Yaskawa INFORM job: MALBEN3.JBI

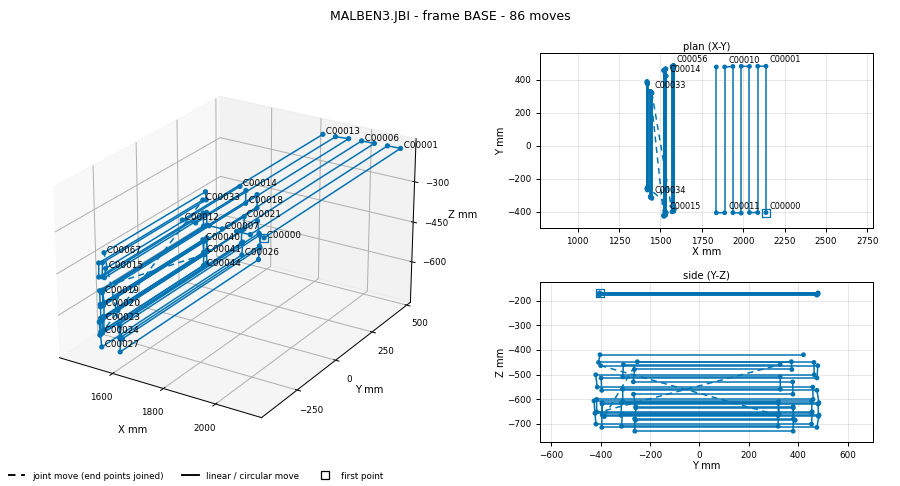
[picture p0: tool path of MALBEN3.JBI in frame BASE, 86 of 92 moves have a stored position in this frame; points joined in program order, loops and branches not executed]
/JOB
//NAME MALBEN3
//POS
///NPOS 86,0,86,0,0,0
///TOOL 0
///POSTYPE BASE
///RECTAN
///RCONF 1,0,0,0,0,0,0,0,0,0,0,0,0,0,0,0,0,0,0,0,0,0,0,0
C00000=2138.089252,-404.380452,-169.043680,175.000000,5.000000,5.000000
C00001=2138.089252,480.563343,-169.043680,175.000000,5.000000,5.000000
C00002=2088.089252,480.435732,-170.096495,175.000000,5.000000,5.000000
C00003=2088.089252,-404.293829,-170.096495,175.000000,5.000000,5.000000
C00004=2038.089252,-404.161569,-171.304879,175.000000,5.000000,5.000000
C00005=2038.089252,479.548369,-171.304879,175.000000,5.000000,5.000000
C00006=1988.089252,480.242625,-172.720240,175.000000,5.000000,5.000000
C00007=1988.089252,-407.599887,-172.720240,175.000000,5.000000,5.000000
C00008=1938.089252,-404.906531,-174.491375,175.000000,5.000000,5.000000
C00009=1938.089252,479.135112,-174.491375,175.000000,5.000000,5.000000
C00010=1888.089252,475.934269,-176.316370,175.000000,5.000000,5.000000
C00011=1888.089252,-405.530643,-176.316370,175.000000,5.000000,5.000000
C00012=1837.950754,-405.573743,-177.808492,175.000000,5.000000,5.000000
C00013=1837.950754,475.917367,-177.808492,175.000000,5.000000,5.000000
C00014=1534.901840,421.478015,-419.338167,175.000000,-89.999999,5.000000
C00015=1534.901840,-402.937946,-419.338167,175.000000,-89.999999,5.000000
C00016=1533.144001,-408.647490,-450.491085,175.000000,-89.999999,5.000000
C00017=1533.144001,464.153807,-450.491085,175.000000,-89.999999,5.000000
C00018=1531.375428,464.936799,-500.491085,175.000000,-89.999999,5.000000
C00019=1531.375428,-420.046716,-500.491085,175.000000,-89.999999,5.000000
C00020=1529.352914,-413.942085,-550.491085,175.000000,-89.999999,5.000000
C00021=1529.352914,459.233172,-550.491085,175.000000,-89.999999,5.000000
C00022=1526.912057,460.521115,-600.491085,175.000000,-89.999999,5.000000
C00023=1526.912057,-416.386557,-600.491085,175.000000,-89.999999,5.000000
C00024=1524.500347,-416.295497,-650.491085,175.000000,-89.999999,5.000000
C00025=1524.500347,456.784052,-650.491085,175.000000,-89.999999,5.000000
C00026=1522.504336,454.310846,-700.491085,175.000000,-89.999999,5.000000
C00027=1522.504336,-419.163579,-700.491085,175.000000,-89.999999,5.000000
C00028=1520.880267,-427.203082,-606.153518,180.000000,-60.000000,0.000000
C00029=1520.880267,455.493151,-606.153518,180.000000,-60.000000,0.000000
C00030=1519.374249,455.436528,-656.153518,180.000000,-60.000000,0.000000
C00031=1519.374249,-422.503865,-656.153518,180.000000,-60.000000,0.000000
C00032=1519.374249,-422.503865,-656.153518,180.000000,-60.000000,0.000000
C00033=1438.715086,327.474473,-459.345178,175.000000,-89.999999,5.000000
C00034=1438.715086,-307.755951,-459.345178,175.000000,-89.999999,5.000000
C00035=1439.798940,-310.872345,-509.345178,175.000000,-89.999999,5.000000
C00036=1439.798940,327.369569,-509.345178,175.000000,-89.999999,5.000000
C00037=1441.037287,327.734598,-559.345178,175.000000,-89.999999,5.000000
C00038=1441.037287,-310.730484,-559.345178,175.000000,-89.999999,5.000000
C00039=1442.396814,-310.620464,-609.345178,175.000000,-89.999999,5.000000
C00040=1442.396814,320.382842,-609.345178,175.000000,-89.999999,5.000000
C00041=1443.632843,322.978132,-659.345178,175.000000,-89.999999,5.000000
C00042=1443.632843,-311.906310,-659.345178,175.000000,-89.999999,5.000000
C00043=1445.183093,-315.667760,-709.345178,175.000000,-89.999999,5.000000
C00044=1445.183093,319.105240,-709.345178,175.000000,-89.999999,5.000000
C00045=1446.831419,319.750011,-615.007611,180.000000,-60.000000,0.000000
C00046=1446.831419,-315.758164,-615.007611,180.000000,-60.000000,0.000000
C00047=1448.220568,-317.504562,-665.007611,180.000000,-60.000000,0.000000
C00048=1448.220568,318.562813,-665.007611,180.000000,-60.000000,0.000000
C00049=1448.220568,318.562813,-665.007611,180.000000,-60.000000,0.000000
C00050=1570.356830,-399.922593,-463.648284,175.000000,-89.999999,5.000000
C00051=1570.356830,479.704633,-463.648284,175.000000,-89.999999,5.000000
C00052=1572.586404,476.504213,-513.648284,175.000000,-89.999999,5.000000
C00053=1572.586404,-398.280973,-513.648284,175.000000,-89.999999,5.000000
C00054=1574.691641,-395.744807,-563.648284,175.000000,-89.999999,5.000000
C00055=1574.691641,476.324205,-563.648284,175.000000,-89.999999,5.000000
C00056=1576.436703,484.068766,-613.648284,175.000000,-89.999999,5.000000
C00057=1576.436703,-394.544332,-613.648284,175.000000,-89.999999,5.000000
C00058=1578.039943,-393.977688,-663.648284,175.000000,-89.999999,5.000000
C00059=1578.039943,484.690765,-663.648284,175.000000,-89.999999,5.000000
C00060=1579.649911,475.998417,-713.648284,175.000000,-89.999999,5.000000
C00061=1579.649911,-395.540713,-713.648284,175.000000,-89.999999,5.000000
C00062=1580.841793,-394.570108,-619.310716,180.000000,-60.000000,0.000000
C00063=1580.841793,480.898770,-619.310716,180.000000,-60.000000,0.000000
C00064=1582.269908,482.315169,-669.310716,180.000000,-60.000000,0.000000
C00065=1582.269908,-385.635636,-669.310716,180.000000,-60.000000,0.000000
C00066=1582.269908,-385.635636,-669.310716,180.000000,-60.000000,0.000000
C00067=1420.964910,-251.559719,-447.665037,175.000000,-89.999999,5.000000
C00068=1420.964910,372.604123,-447.665037,175.000000,-89.999999,5.000000
C00069=1422.373131,374.697923,-479.185471,175.000000,-89.999999,5.000000
C00070=1422.373131,-263.019191,-479.185471,175.000000,-89.999999,5.000000
C00071=1421.975445,-267.696341,-529.185471,175.000000,-89.999999,5.000000
C00072=1421.975445,377.834218,-529.185471,175.000000,-89.999999,5.000000
C00073=1421.594266,378.934991,-579.185471,175.000000,-89.999999,5.000000
C00074=1421.594266,-266.992153,-579.185471,175.000000,-89.999999,5.000000
C00075=1420.418300,-258.080778,-629.185471,175.000000,-89.999999,5.000000
C00076=1420.418300,379.690351,-629.185471,175.000000,-89.999999,5.000000
C00077=1419.981840,380.884372,-679.185471,175.000000,-89.999999,5.000000
C00078=1419.981840,-262.435258,-679.185471,175.000000,-89.999999,5.000000
C00079=1419.737986,-261.680466,-729.185471,175.000000,-89.999999,5.000000
C00080=1419.737986,379.769100,-729.185471,175.000000,-89.999999,5.000000
C00081=1419.270374,380.316359,-634.847904,180.000000,-60.000000,0.000000
C00082=1419.270374,-257.794213,-634.847904,180.000000,-60.000000,0.000000
C00083=1418.737426,-258.418231,-684.847904,180.000000,-60.000000,0.000000
C00084=1418.737426,387.426469,-684.847904,180.000000,-60.000000,0.000000
C00085=1418.737426,387.426469,-684.847904,180.000000,-60.000000,0.000000
///POSTYPE PULSE
///PULSE
EC00000=0
EC00001=0
EC00002=0
EC00003=0
EC00004=0
EC00005=0
EC00006=0
EC00007=0
EC00008=0
EC00009=0
EC00010=0
EC00011=0
EC00012=0
EC00013=0
EC00014=0
EC00015=0
EC00016=0
EC00017=0
EC00018=0
EC00019=0
EC00020=0
EC00021=0
EC00022=0
EC00023=0
EC00024=0
EC00025=0
EC00026=0
EC00027=0
EC00028=0
EC00029=0
EC00030=0
EC00031=0
EC00032=92160
EC00033=92160
EC00034=92160
EC00035=92160
EC00036=92160
EC00037=92160
EC00038=92160
EC00039=92160
EC00040=92160
EC00041=92160
EC00042=92160
EC00043=92160
EC00044=92160
EC00045=92160
EC00046=92160
EC00047=92160
EC00048=92160
EC00049=184320
EC00050=184320
EC00051=184320
EC00052=184320
EC00053=184320
EC00054=184320
EC00055=184320
EC00056=184320
EC00057=184320
EC00058=184320
EC00059=184320
EC00060=184320
EC00061=184320
EC00062=184320
EC00063=184320
EC00064=184320
EC00065=184320
EC00066=276480
EC00067=276480
EC00068=276480
EC00069=276480
EC00070=276480
EC00071=276480
EC00072=276480
EC00073=276480
EC00074=276480
EC00075=276480
EC00076=276480
EC00077=276480
EC00078=276480
EC00079=276480
EC00080=276480
EC00081=276480
EC00082=276480
EC00083=276480
EC00084=276480
EC00085=368640
//INST
///DATE 2023/03/16 10:48
///ATTR SC,RW,RJ
////FRAME BASE
///GROUP1 RB1,ST1
NOP
MOVJ P009 EX000 VJ=15.00
MOVJ C00000 EC00000 VJ=15.0
CALL JOB:SPYON
MOVL C00001 EC00001 V=300.0
MOVL C00002 EC00002 V=300.0
MOVL C00003 EC00003 V=300.0
MOVL C00004 EC00004 V=300.0
MOVL C00005 EC00005 V=300.0
MOVL C00006 EC00006 V=300.0
MOVL C00007 EC00007 V=300.0
MOVL C00008 EC00008 V=300.0
MOVL C00009 EC00009 V=300.0
MOVL C00010 EC00010 V=300.0
MOVL C00011 EC00011 V=300.0
MOVL C00012 EC00012 V=300.0
MOVL C00013 EC00013 V=300.0
CALL JOB:SPYOF
MOVJ P009 VJ=15.00
MOVJ C00014 EC00014 VJ=15.0
CALL JOB:SPYON
MOVL C00015 EC00015 V=300.0
MOVL C00016 EC00016 V=300.0
MOVL C00017 EC00017 V=300.0
MOVL C00018 EC00018 V=300.0
MOVL C00019 EC00019 V=300.0
MOVL C00020 EC00020 V=300.0
MOVL C00021 EC00021 V=300.0
MOVL C00022 EC00022 V=300.0
MOVL C00023 EC00023 V=300.0
MOVL C00024 EC00024 V=300.0
MOVL C00025 EC00025 V=300.0
MOVL C00026 EC00026 V=300.0
MOVL C00027 EC00027 V=300.0
MOVL C00028 EC00028 V=300.0
MOVL C00029 EC00029 V=300.0
MOVL C00030 EC00030 V=300.0
MOVL C00031 EC00031 V=300.0
CALL JOB:SPYOF
MOVJ P009 VJ=15.00
MOVL C00032 EC00032 V=300.0
MOVJ C00033 EC00033 VJ=15.0
CALL JOB:SPYON
MOVL C00034 EC00034 V=300.0
MOVL C00035 EC00035 V=300.0
MOVL C00036 EC00036 V=300.0
MOVL C00037 EC00037 V=300.0
MOVL C00038 EC00038 V=300.0
MOVL C00039 EC00039 V=300.0
MOVL C00040 EC00040 V=300.0
MOVL C00041 EC00041 V=300.0
MOVL C00042 EC00042 V=300.0
MOVL C00043 EC00043 V=300.0
MOVL C00044 EC00044 V=300.0
MOVL C00045 EC00045 V=300.0
MOVL C00046 EC00046 V=300.0
MOVL C00047 EC00047 V=300.0
MOVL C00048 EC00048 V=300.0
CALL JOB:SPYOF
MOVJ P009 VJ=15.00
MOVL C00049 EC00049 V=300.0
MOVJ C00050 EC00050 VJ=15.0
CALL JOB:SPYON
MOVL C00051 EC00051 V=300.0
MOVL C00052 EC00052 V=300.0
MOVL C00053 EC00053 V=300.0
MOVL C00054 EC00054 V=300.0
MOVL C00055 EC00055 V=300.0
MOVL C00056 EC00056 V=300.0
MOVL C00057 EC00057 V=300.0
MOVL C00058 EC00058 V=300.0
MOVL C00059 EC00059 V=300.0
MOVL C00060 EC00060 V=300.0
MOVL C00061 EC00061 V=300.0
MOVL C00062 EC00062 V=300.0
MOVL C00063 EC00063 V=300.0
MOVL C00064 EC00064 V=300.0
MOVL C00065 EC00065 V=300.0
CALL JOB:SPYOF
MOVJ P009 VJ=15.00
MOVL C00066 EC00066 V=300.0
MOVJ C00067 EC00067 VJ=15.0
CALL JOB:SPYON
MOVL C00068 EC00068 V=300.0
MOVL C00069 EC00069 V=300.0
MOVL C00070 EC00070 V=300.0
MOVL C00071 EC00071 V=300.0
MOVL C00072 EC00072 V=300.0
MOVL C00073 EC00073 V=300.0
MOVL C00074 EC00074 V=300.0
MOVL C00075 EC00075 V=300.0
MOVL C00076 EC00076 V=300.0
MOVL C00077 EC00077 V=300.0
MOVL C00078 EC00078 V=300.0
MOVL C00079 EC00079 V=300.0
MOVL C00080 EC00080 V=300.0
MOVL C00081 EC00081 V=300.0
MOVL C00082 EC00082 V=300.0
MOVL C00083 EC00083 V=300.0
MOVL C00084 EC00084 V=300.0
CALL JOB:SPYOF
MOVJ P009 VJ=15.00
MOVL C00085 EC00085 V=300.0
END
